{attribute 'qualified_only'}
//{attribute 'strict'}
TYPE eNetworkState :
(
	unknown := 0,
	searching := 1,
	Unregistered := 2,
	Registered := 3,
	Roaming := 4
	);
END_TYPE

(* stored: Version 1.1.0.1, ProductVersion 3.1.4026.18
   DUT eNetworkState: Id {4779bd32-343e-4a22-b2e0-c70e7c17caba} *)
